PROGRAM MAIN
VAR
END_VAR

Echange_OPCUA();

END_PROGRAM

(* stored: Version 1.1.0.1, ProductVersion 3.1.4026.18
   POU MAIN: Id {513fc92b-fdea-4ce5-9d3a-424fa6b6b858}, SpecialFunc None *)
